// MUST be in same order and number as AlarmSignals
TYPE AlarmsDelaysB :
STRUCT
	RegulationDeviation: TIME := T#60M;
	SupplyAirDeviation: TIME := T#60M;
	ExtractAirDeviation: TIME := T#60M;
	SupplyFan: TIME := T#60S;
	ExtractFan: TIME := T#60S;
	HeatExchangerEfficiency: TIME := T#1H;
	Defrost: TIME := T#5S;
	SupplyFilter: TIME := T#1H;
	ExtractFilter: TIME := T#1H;
	SmokeDetectorServiceSupply: TIME := T#5S;
	SmokeDetectorServiceExtract: TIME := T#5S;
	Pump1: TIME := T#5S;
	Pump2: TIME := T#5S;
	DamperError: TIME := T#30S;
	CommunicationError: TIME := T#30S;
	DamperModuleService: TIME := T#5S;
	Tx1Fail: TIME := T#1M;
END_STRUCT
END_TYPE

(* stored: Version 1.1.0.1, ProductVersion 3.1.4024.6
   DUT AlarmsDelaysB: Id {809e6806-49a9-41d0-b284-3f497d289f53} *)
